FUNCTION_BLOCK ArgoTx (* goFB_ignore *)
  (* Standard: 61499-2 *)
  (* Version 0.1, 2017-00-09, hpea485, UOA *)
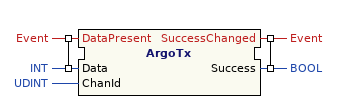
  EVENT_INPUT
    DataPresent WITH Data;
  END_EVENT
  EVENT_OUTPUT
    SuccessChanged WITH Success;
  END_EVENT
  VAR_INPUT
    Data : INT;
    ChanId : UDINT;
  END_VAR
  VAR_OUTPUT
    Success : BOOL;
  END_VAR
  EC_STATES
    Start;
  END_STATES
END_FUNCTION_BLOCK
